{attribute 'linkalways'} 
{attribute 'no_explicit_call' := 'This FB is a CLASS and must be accessed using methods or properties'}
{attribute 'enable_dynamic_creation'}
FUNCTION_BLOCK FINAL LT_SINT EXTENDS Node
VAR
	in1 : _SINT(0);
	in2 : _SINT(0);
	out : _BOOL(FALSE);
END_VAR

METHOD PUBLIC Clone : I_Node
VAR
	pNode : POINTER TO LT_SINT;
END_VAR
pNode := __NEW(LT_SINT);
Clone := pNode^;
END_METHOD

METHOD FB_init : BOOL
VAR_INPUT
	bInitRetains : BOOL; // if TRUE, the retain variables are initialized (warm start / cold start)
	bInCopyCode : BOOL;  // if TRUE, the instance afterwards gets moved into the copy code (online change)
END_VAR
AddInput('in1',THIS^.in1);
AddInput('in2',THIS^.in2);
AddOutput('out', THIS^.out);
END_METHOD

METHOD PROTECTED OnExecute
VAR
END_VAR
out.Value := in1.Value < in2.Value;
END_METHOD

END_FUNCTION_BLOCK

(* stored: Version 1.1.0.1, ProductVersion 3.1.4024.15
   POU LT_SINT: Id {40ce4995-7a16-4a80-87de-d729c21d4bf9}, SpecialFunc None
   Folder Constructor: Id {f42baab1-3059-4c64-8b5f-21202cb462aa}
   Method Clone: Id {4db85f2d-77a5-4bc0-87bb-38d2bfaf120a}
   Method FB_init: Id {1e635308-6795-4eb2-b15e-4e6a876d4317}
   Method OnExecute: Id {dca8c885-1fb6-4f0c-bd24-6242ff99a034} *)
